Staubli VAL3: onRun.pgx

public program onRun(string& x_sItem[])
  local num l_nValue
  local bool l_bOk
begin
  //
  // convert to a num
  l_bOk=true
  toNum(x_sItem,l_nValue,l_bOk)
   // NB the robot will no STOP
  delay(l_nValue)
  //
end
